{attribute addProperty BoxType "ELX9560-0000-0018"}
{attribute addProperty Id "Uex_OKAT %I*BOOL81"}
{attribute addProperty CRC "2749195422"}
{attribute addProperty SizeInBites "8"}
{attribute addProperty SizeInBytes "1"}
TYPE Status_Uex_A3DD649E :
STRUCT
	{attribute addProperty Name "Uex_OK"}
	Uex_OK AT %I* : BOOL;
END_STRUCT
END_TYPE

(* stored: Version 1.2.0.0, ProductVersion 3.1.4024.9
   DUT Status_Uex_A3DD649E: Id {55b82801-4078-46b6-9478-3aeea9835a6a} *)
